{attribute addProperty BoxType "CU1128-0000-0002"}
{attribute addProperty Id "A_0007_CU1521_0010_0000CU1521_179A0949162A_0008_CU1561_0000_0000CU1561_179A0949162A_0009_CU2508_0000_0000CU2508_179A0949162A_0010_CU2508_0000_0016CU2508_194A340D8010A_0011_CU2508_0000_0017CU2508_36DE295224230.25A_0012_CU2508_0000_0018CU2508_36DE295224230.25A_0013_CU2508_0000_0019CU2508_36DE295224230.25A_0006_CU1128_0000_0002_2_CU1128_BCU1128_179A0949162A_0006_CU1128_0000_0002_3_CU1128_CCU1128_179A0949162"}
{attribute addProperty CRC "230028729"}
{attribute addProperty SizeInBites "886"}
{attribute addProperty SizeInBytes "110.75"}
TYPE A_0006_CU1128_0000_0002_0DB5F5B9 EXTENDS CU1128_179A0949 :
STRUCT
	{attribute addProperty Name "A_0007_CU1521_0010_0000"}
	A_0007_CU1521_0010_0000 : CU1521_179A0949;
	{attribute addProperty Name "A_0008_CU1561_0000_0000"}
	A_0008_CU1561_0000_0000 : CU1561_179A0949;
	{attribute addProperty Name "A_0009_CU2508_0000_0000"}
	A_0009_CU2508_0000_0000 : CU2508_179A0949;
	{attribute addProperty Name "A_0010_CU2508_0000_0016"}
	A_0010_CU2508_0000_0016 : CU2508_194A340D;
	{attribute addProperty Name "A_0011_CU2508_0000_0017"}
	A_0011_CU2508_0000_0017 : CU2508_36DE2952;
	{attribute addProperty Name "A_0012_CU2508_0000_0018"}
	A_0012_CU2508_0000_0018 : CU2508_36DE2952;
	{attribute addProperty Name "A_0013_CU2508_0000_0019"}
	A_0013_CU2508_0000_0019 : CU2508_36DE2952;
	{attribute addProperty Name "A_0006_CU1128_0000_0002_2_CU1128_B"}
	A_0006_CU1128_0000_0002_2_CU1128_B : CU1128_179A0949;
	{attribute addProperty Name "A_0006_CU1128_0000_0002_3_CU1128_C"}
	A_0006_CU1128_0000_0002_3_CU1128_C : CU1128_179A0949;
END_STRUCT
END_TYPE

(* stored: Version 1.2.0.0, ProductVersion 3.1.4024.9
   DUT A_0006_CU1128_0000_0002_0DB5F5B9: Id {47b0e5e8-2596-49f9-a9e9-d8acfcb1d7b7} *)
